TYPE ST_SafetyAliasOutput :
STRUCT
	sName : STRING; //Name descriptor for the safety output
    bState : BOOL;
END_STRUCT
END_TYPE

(* stored: Version 1.1.0.1, ProductVersion 3.1.4024.11
   DUT ST_SafetyAliasOutput: Id {8a85b2a5-61fa-4f89-9d55-2acad09a8c3a} *)
